FUNCTION F_GetZoneErrorData : ST_ZoneErrorStruct
(**************************************************************************************
 * 	Application		:	BoxControl Framework
 *	Revision		:	$Revision: 404529 $
 *	Revision date	:	$Date: 2018-04-23 08:21:38 +0200 (Mo., 23 Apr 2018) $
 *	Last changed by	:	$Author: b7bolm $
 *	URL				:	$URL: http://almscdc.swisslog.com/repo/SWPD/Development/BoxControlFramework/20_Release/trunk/01_Software/BCF/BCF/JumpStart/20_Product/10_App/12_E_Functions/10_Lib/10_Conv/10_Functions/F_GetZoneErrorData.TcPOU $
 *
 *	Purpose			:	Return zone error data
 *
 * ------------------------------------------------------------------------------------
 *	Copyright Swisslog [IP AG], Switzerland. All rights reserved.
 * 
 * ------------------------------------------------------------------------------------
 *	
 * 	Revision History: 
 *
 * 	VERSION			DATE			INITIALS			DESCRIPTION
 *	0.1				01.01.2001		swl					Example
 *
 **************************************************************************************)
VAR_INPUT
	eFunctionNumber		: E_FunctionNumber;
	ZoneNumber			: INT; 
END_VAR
VAR
	ZoneData			: ARRAY[1..NUMBER_OF_ZONES_PER_FUNCTION] OF ST_ZoneData; // all zone data
END_VAR


// Check if function number and zone is valid
IF eFunctionNumber > E_FunctionNumber.F_BEGIN_FUNCTION AND
   eFunctionNumber < E_FunctionNumber.F_END_FUNCTION AND
   ZoneNumber > 0 AND ZoneNumber <= NUMBER_OF_ZONES_PER_FUNCTION THEN
  
   IF __ISVALIDREF(FunctionRegistry[eFunctionNumber].Zone[ZoneNumber].refZoneData) THEN
		// Zone errordata
		F_GetZoneErrorData := FunctionRegistry[eFunctionNumber].Zone[ZoneNumber].refZoneData.ErrorData;
	END_IF
END_IF

END_FUNCTION

(* stored: Version 1.1.0.1, ProductVersion 3.1.4022.12
   POU F_GetZoneErrorData: Id {ce342298-13fd-4de6-8139-057dfab667c7}, SpecialFunc None *)
